// TIA Portal V20 export
FUNCTION_BLOCK "TestIo"   // FB306, FBD
{ S7_Optimized_Access := 'TRUE' }
// stored: AutoNumber false, MemoryReserve 100, SetENOAutomatically false
BEGIN

REGION Network 1 (SCL): Data PLC Input Normal

   "ComSd".Data.PlcInputNormal."I0.0" := "I_IN1_EXT+SGV";
   "ComSd".Data.PlcInputNormal."I0.1" := "I_IN2_EXT+SGV";
   "ComSd".Data.PlcInputNormal."I0.2" := "I_IN3_EXT+SGV";
   "ComSd".Data.PlcInputNormal."I0.3" := "I_0E1+SGV";
   "ComSd".Data.PlcInputNormal."I0.4" := "I_0E2+SGX";
   "ComSd".Data.PlcInputNormal."I0.5" := "I_0F1.1+SGV";
   "ComSd".Data.PlcInputNormal."I0.6" := "I_0SH1+SSTR";
   "ComSd".Data.PlcInputNormal."I0.7" := "I_14SB0+HMI";
   "ComSd".Data.PlcInputNormal."I1.0" := "I_14SB1+HMI";
   "ComSd".Data.PlcInputNormal."I1.1" := "I_8S1.T_in";
   "ComSd".Data.PlcInputNormal."I1.2" := "I_8S2.T_out";
   "ComSd".Data.PlcInputNormal."I1.3" := "I_8S1.L_in";
   "ComSd".Data.PlcInputNormal."I1.4" := "I_8S2.L_out";
   "ComSd".Data.PlcInputNormal."I1.5" := "I_8S1.R_in";
   "ComSd".Data.PlcInputNormal."I1.6" := "I_8S2.R_out";
   "ComSd".Data.PlcInputNormal."I1.7" := "I_1BTR2+SGV";
   "ComSd".Data.PlcInputNormal."I2.0" := "I_8S1.B_left";
   "ComSd".Data.PlcInputNormal."I2.1" := "I_8S2.B_right";
   "ComSd".Data.PlcInputNormal."I2.2" := "I_1BTR2+SGX";
   "ComSd".Data.PlcInputNormal."I2.3" := "I_0E1.1+SGV";
   "ComSd".Data.PlcInputNormal."I2.4" := "I_spare24";
   "ComSd".Data.PlcInputNormal."I2.5" := "I_spare25";
   "ComSd".Data.PlcInputNormal."I2.6" := "I_spare26";
   "ComSd".Data.PlcInputNormal."I2.7" := "I_spare27";
END_REGION

REGION Network 2 (SCL): Data PLC Input Safety

   "ComSd".Data.PlcInputSafety."I800.0" := "SI_NA_EXT+SGV";
   "ComSd".Data.PlcInputSafety."I800.1" := "SI_14SB0/1+HMI";
   "ComSd".Data.PlcInputSafety."I800.2" := "SI_14SB1+SSTL";
   "ComSd".Data.PlcInputSafety."I800.3" := "SI_14SB2+SSTL";
   "ComSd".Data.PlcInputSafety."I808.0" := "SI_14SS1.TL+SGV";
   "ComSd".Data.PlcInputSafety."I808.1" := "SI_14SS1.BL+SGV";
   "ComSd".Data.PlcInputSafety."I808.2" := "SI_14SS1.TR+SGV";
   "ComSd".Data.PlcInputSafety."I808.3" := "SI_14SS1.BR+SGV";
   "ComSd".Data.PlcInputSafety."I816.0" := "SI_14SS1.TL+SGX";
   "ComSd".Data.PlcInputSafety."I816.1" := "SI_14SS1.BL+SGX";
   "ComSd".Data.PlcInputSafety."I816.2" := "SI_14SS1.TR+SGX";
   "ComSd".Data.PlcInputSafety."I816.3" := "SI_14SS1.BR+SGX";
   "ComSd".Data.PlcInputSafety."I824.0" := "SI_8U1+SGV";
   "ComSd".Data.PlcInputSafety."I824.1" := "SI_14KA1+SGV";
   "ComSd".Data.PlcInputSafety."I824.2" := "SI_14KA2+SGV";
   "ComSd".Data.PlcInputSafety."I824.3" := "SI_5AX1+SGX";
END_REGION

REGION Network 3 (SCL): Data PLC Output Normal

   "ComSd".Data.PlcOutputNormal."Q0.0" := "O_14VK1+SGV";
   "ComSd".Data.PlcOutputNormal."Q0.1" := "O_14VK2+SGV";
   "ComSd".Data.PlcOutputNormal."Q0.2" := "O_0VK1+SGV";
   "ComSd".Data.PlcOutputNormal."Q0.3" := "O_0VK2+SGV";
   "ComSd".Data.PlcOutputNormal."Q0.4" := "O_0VK3+SGV";
   "ComSd".Data.PlcOutputNormal."Q0.5" := "O_0VK4+SGV";
   "ComSd".Data.PlcOutputNormal."Q0.6" := "O_0F1.1+SGV";
   "ComSd".Data.PlcOutputNormal."Q0.7" := "O_0KA0.1+SGV";
   "ComSd".Data.PlcOutputNormal."Q1.0" := "O_0KA0.2+SGV";
   "ComSd".Data.PlcOutputNormal."Q1.1" := "O_0KA1+SGV";
   "ComSd".Data.PlcOutputNormal."Q1.2" := "O_8M1.T_c";
   "ComSd".Data.PlcOutputNormal."Q1.3" := "O_8M1.T_o";
   "ComSd".Data.PlcOutputNormal."Q1.4" := "O_8M1.L_c";
   "ComSd".Data.PlcOutputNormal."Q1.5" := "O_8M1.L_o";
   "ComSd".Data.PlcOutputNormal."Q1.6" := "O_8M1.R_c";
   "ComSd".Data.PlcOutputNormal."Q1.7" := "O_8M1.R_o";
   "ComSd".Data.PlcOutputNormal."Q2.0" := "O_8KA1+SGV";
   "ComSd".Data.PlcOutputNormal."Q2.1" := "O_8M1.B_l";
   "ComSd".Data.PlcOutputNormal."Q2.2" := "O_8M1.B_r";
   "ComSd".Data.PlcOutputNormal."Q2.3" := "O_2YV1/2.B+SGV";
   "ComSd".Data.PlcOutputNormal."Q2.4" := "O_2YV1.L+SGV";
   "ComSd".Data.PlcOutputNormal."Q2.5" := "O_2YV1.R+SGV";
   "ComSd".Data.PlcOutputNormal."Q2.6" := "O_5YV1+SGX";
   "ComSd".Data.PlcOutputNormal."Q2.7" := "O_spare27";
END_REGION

REGION Network 4 (SCL): Data PLC Output Safety

   "ComSd".Data.PlcOutputSafety."Q900.0" := "SO_safetynew";
   "ComSd".Data.PlcOutputSafety."Q900.1" := "SO_14HV1+SSTL/R";
   "ComSd".Data.PlcOutputSafety."Q900.2" := "SO_14KA1+SGV";
   "ComSd".Data.PlcOutputSafety."Q900.3" := "SO_14KA2+SGV";
   "ComSd".Data.PlcOutputSafety."Q908.0" := "SO_ST.3HF+SGV";
   "ComSd".Data.PlcOutputSafety."Q908.1" := "SO_ST.5HF+SGV";
   "ComSd".Data.PlcOutputSafety."Q908.2" := "SO_5AX1+SGX";
   "ComSd".Data.PlcOutputSafety."Q908.3" := "SO_spare9083";
END_REGION
END_FUNCTION_BLOCK
